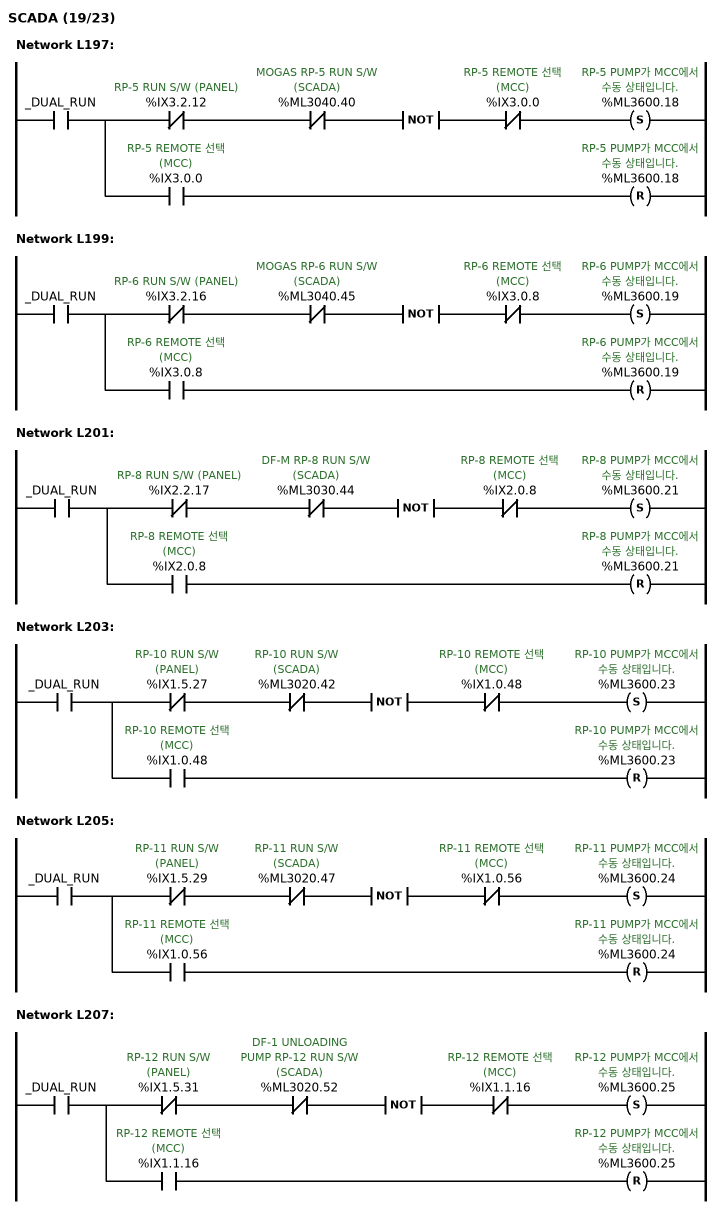
(* [picture p72: SCADA rungs L197-L207] *)
(* Rung L197 *)
IF NOT (_DUAL_RUN AND NOT %IX3.2.12 AND NOT %ML3040.40) AND NOT %IX3.0.0 THEN %ML3600.18 := TRUE; END_IF;
IF _DUAL_RUN AND %IX3.0.0 THEN %ML3600.18 := FALSE; END_IF;
(* Rung L199 *)
IF NOT (_DUAL_RUN AND NOT %IX3.2.16 AND NOT %ML3040.45) AND NOT %IX3.0.8 THEN %ML3600.19 := TRUE; END_IF;
IF _DUAL_RUN AND %IX3.0.8 THEN %ML3600.19 := FALSE; END_IF;
(* Rung L201 *)
IF NOT (_DUAL_RUN AND NOT %IX2.2.17 AND NOT %ML3030.44) AND NOT %IX2.0.8 THEN %ML3600.21 := TRUE; END_IF;
IF _DUAL_RUN AND %IX2.0.8 THEN %ML3600.21 := FALSE; END_IF;
(* Rung L203 *)
IF NOT (_DUAL_RUN AND NOT %IX1.5.27 AND NOT %ML3020.42) AND NOT %IX1.0.48 THEN %ML3600.23 := TRUE; END_IF;
IF _DUAL_RUN AND %IX1.0.48 THEN %ML3600.23 := FALSE; END_IF;
(* Rung L205 *)
IF NOT (_DUAL_RUN AND NOT %IX1.5.29 AND NOT %ML3020.47) AND NOT %IX1.0.56 THEN %ML3600.24 := TRUE; END_IF;
IF _DUAL_RUN AND %IX1.0.56 THEN %ML3600.24 := FALSE; END_IF;
(* Rung L207 *)
IF NOT (_DUAL_RUN AND NOT %IX1.5.31 AND NOT %ML3020.52) AND NOT %IX1.1.16 THEN %ML3600.25 := TRUE; END_IF;
IF _DUAL_RUN AND %IX1.1.16 THEN %ML3600.25 := FALSE; END_IF;

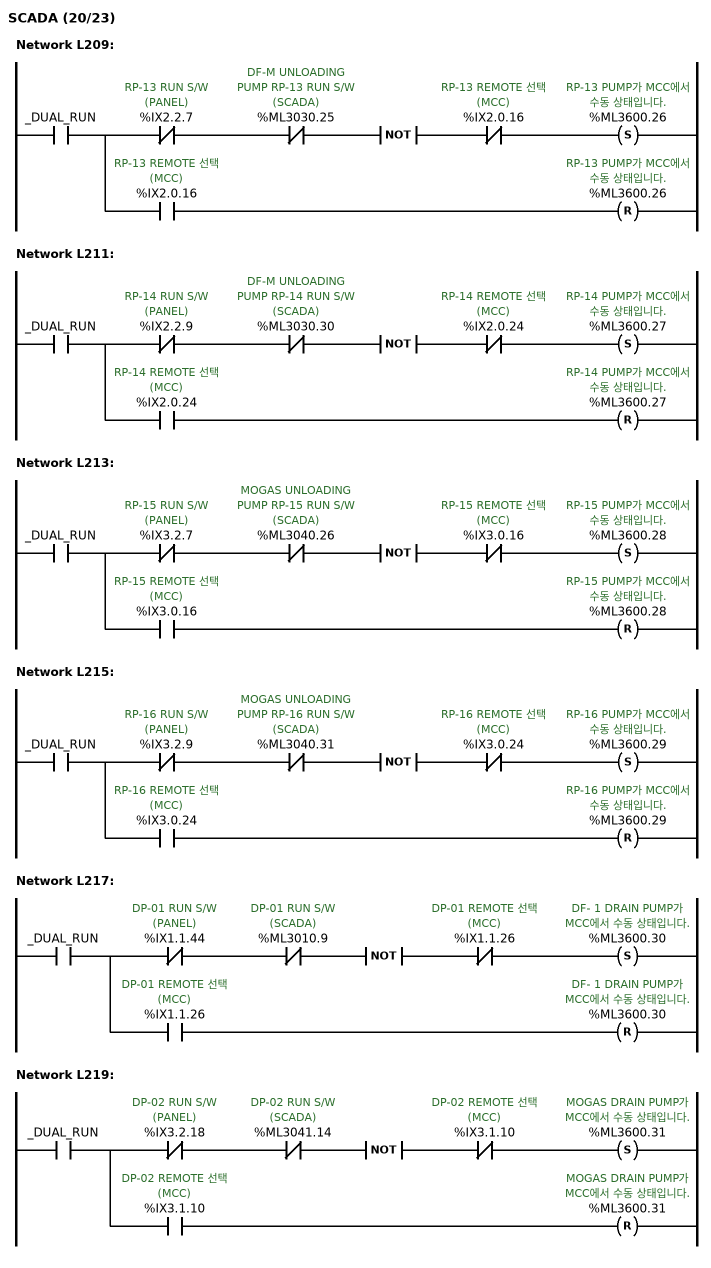
(* Rung L209 *)
IF NOT (_DUAL_RUN AND NOT %IX2.2.7 AND NOT %ML3030.25) AND NOT %IX2.0.16 THEN %ML3600.26 := TRUE; END_IF;
IF _DUAL_RUN AND %IX2.0.16 THEN %ML3600.26 := FALSE; END_IF;
(* Rung L211 *)
IF NOT (_DUAL_RUN AND NOT %IX2.2.9 AND NOT %ML3030.30) AND NOT %IX2.0.24 THEN %ML3600.27 := TRUE; END_IF;
IF _DUAL_RUN AND %IX2.0.24 THEN %ML3600.27 := FALSE; END_IF;
(* Rung L213 *)
IF NOT (_DUAL_RUN AND NOT %IX3.2.7 AND NOT %ML3040.26) AND NOT %IX3.0.16 THEN %ML3600.28 := TRUE; END_IF;
IF _DUAL_RUN AND %IX3.0.16 THEN %ML3600.28 := FALSE; END_IF;
(* Rung L215 *)
IF NOT (_DUAL_RUN AND NOT %IX3.2.9 AND NOT %ML3040.31) AND NOT %IX3.0.24 THEN %ML3600.29 := TRUE; END_IF;
IF _DUAL_RUN AND %IX3.0.24 THEN %ML3600.29 := FALSE; END_IF;
(* Rung L217 *)
IF NOT (_DUAL_RUN AND NOT %IX1.1.44 AND NOT %ML3010.9) AND NOT %IX1.1.26 THEN %ML3600.30 := TRUE; END_IF;
IF _DUAL_RUN AND %IX1.1.26 THEN %ML3600.30 := FALSE; END_IF;
(* Rung L219 *)
IF NOT (_DUAL_RUN AND NOT %IX3.2.18 AND NOT %ML3041.14) AND NOT %IX3.1.10 THEN %ML3600.31 := TRUE; END_IF;
IF _DUAL_RUN AND %IX3.1.10 THEN %ML3600.31 := FALSE; END_IF;

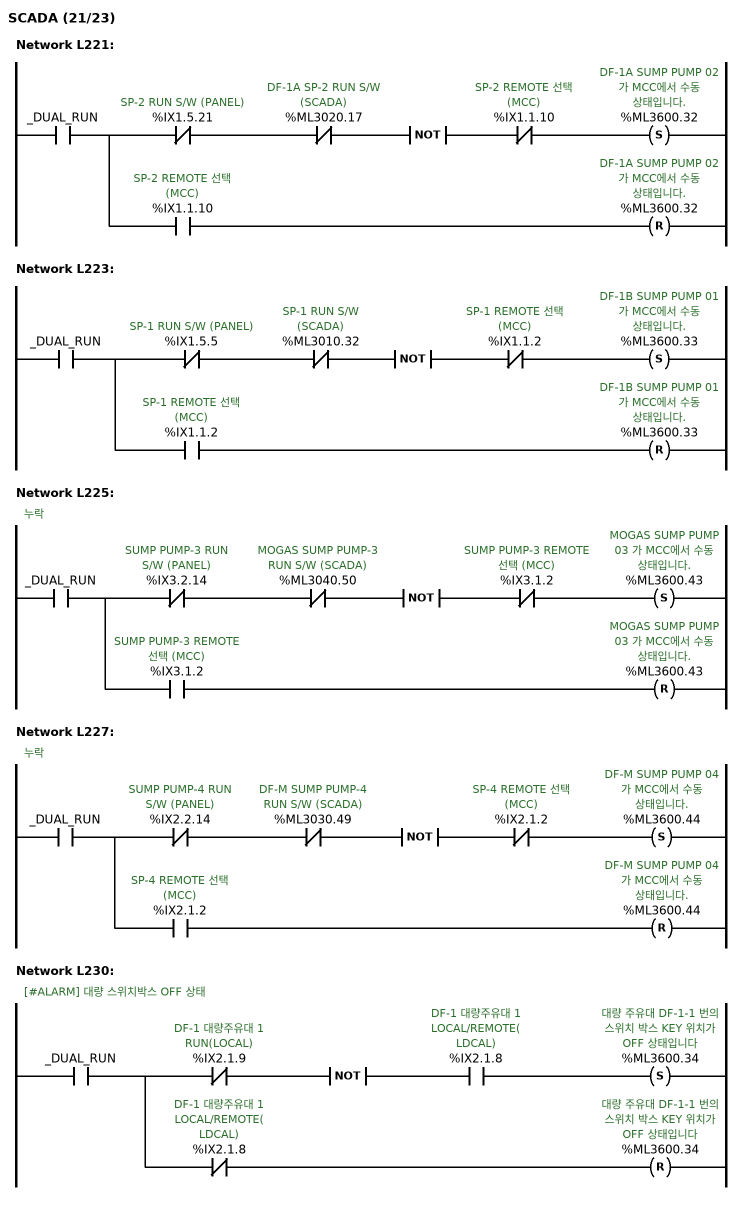
(* Rung L221 *)
IF NOT (_DUAL_RUN AND NOT %IX1.5.21 AND NOT %ML3020.17) AND NOT %IX1.1.10 THEN %ML3600.32 := TRUE; END_IF;
IF _DUAL_RUN AND %IX1.1.10 THEN %ML3600.32 := FALSE; END_IF;
(* Rung L223 *)
IF NOT (_DUAL_RUN AND NOT %IX1.5.5 AND NOT %ML3010.32) AND NOT %IX1.1.2 THEN %ML3600.33 := TRUE; END_IF;
IF _DUAL_RUN AND %IX1.1.2 THEN %ML3600.33 := FALSE; END_IF;
(* Rung L225 *)
IF NOT (_DUAL_RUN AND NOT %IX3.2.14 AND NOT %ML3040.50) AND NOT %IX3.1.2 THEN %ML3600.43 := TRUE; END_IF;
IF _DUAL_RUN AND %IX3.1.2 THEN %ML3600.43 := FALSE; END_IF;
(* 누락 *)
(* Rung L227 *)
IF NOT (_DUAL_RUN AND NOT %IX2.2.14 AND NOT %ML3030.49) AND NOT %IX2.1.2 THEN %ML3600.44 := TRUE; END_IF;
IF _DUAL_RUN AND %IX2.1.2 THEN %ML3600.44 := FALSE; END_IF;
(* 누락 *)
(* [#ALARM] 대량 스위치박스 OFF 상태 *)
(* Rung L230 *)
IF NOT (_DUAL_RUN AND NOT %IX2.1.9) AND %IX2.1.8 THEN %ML3600.34 := TRUE; END_IF;
IF _DUAL_RUN AND NOT %IX2.1.8 THEN %ML3600.34 := FALSE; END_IF;

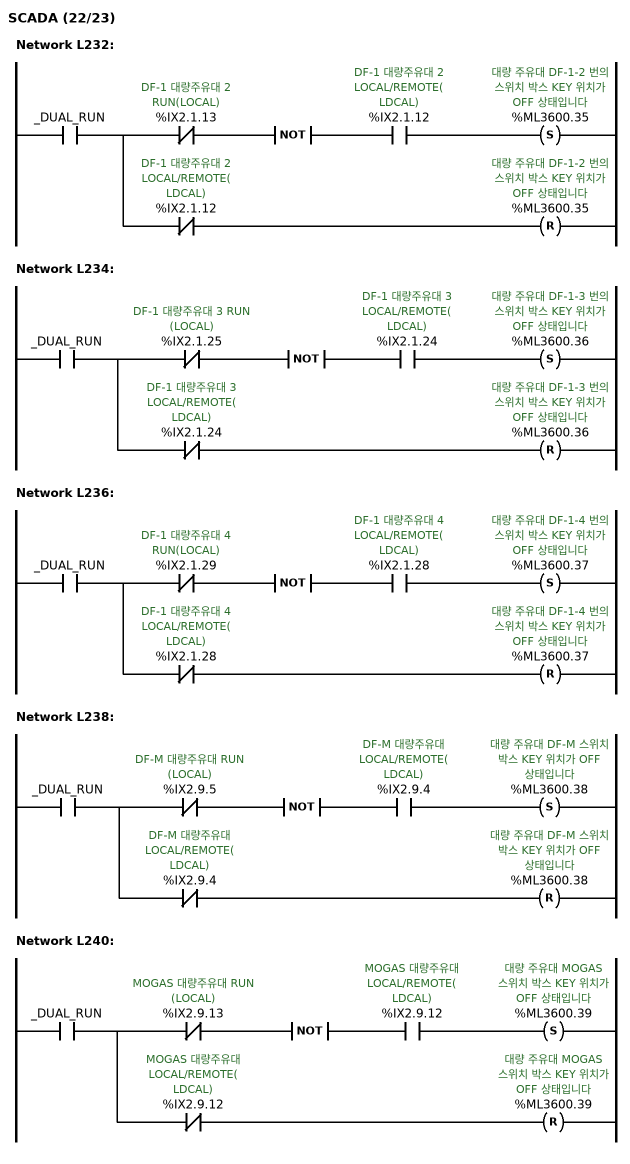
(* Rung L232 *)
IF NOT (_DUAL_RUN AND NOT %IX2.1.13) AND %IX2.1.12 THEN %ML3600.35 := TRUE; END_IF;
IF _DUAL_RUN AND NOT %IX2.1.12 THEN %ML3600.35 := FALSE; END_IF;
(* Rung L234 *)
IF NOT (_DUAL_RUN AND NOT %IX2.1.25) AND %IX2.1.24 THEN %ML3600.36 := TRUE; END_IF;
IF _DUAL_RUN AND NOT %IX2.1.24 THEN %ML3600.36 := FALSE; END_IF;
(* Rung L236 *)
IF NOT (_DUAL_RUN AND NOT %IX2.1.29) AND %IX2.1.28 THEN %ML3600.37 := TRUE; END_IF;
IF _DUAL_RUN AND NOT %IX2.1.28 THEN %ML3600.37 := FALSE; END_IF;
(* Rung L238 *)
IF NOT (_DUAL_RUN AND NOT %IX2.9.5) AND %IX2.9.4 THEN %ML3600.38 := TRUE; END_IF;
IF _DUAL_RUN AND NOT %IX2.9.4 THEN %ML3600.38 := FALSE; END_IF;
(* Rung L240 *)
IF NOT (_DUAL_RUN AND NOT %IX2.9.13) AND %IX2.9.12 THEN %ML3600.39 := TRUE; END_IF;
IF _DUAL_RUN AND NOT %IX2.9.12 THEN %ML3600.39 := FALSE; END_IF;

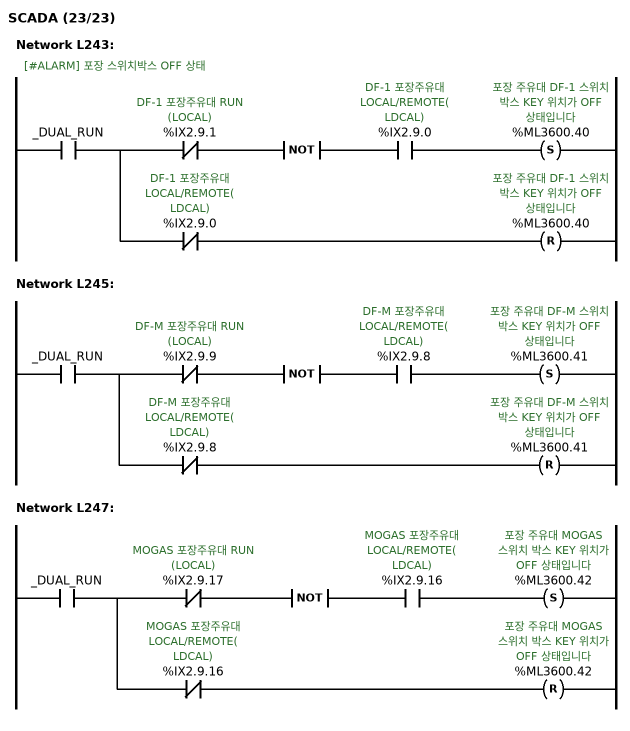
(* [#ALARM] 포장 스위치박스 OFF 상태 *)
(* Rung L243 *)
IF NOT (_DUAL_RUN AND NOT %IX2.9.1) AND %IX2.9.0 THEN %ML3600.40 := TRUE; END_IF;
IF _DUAL_RUN AND NOT %IX2.9.0 THEN %ML3600.40 := FALSE; END_IF;
(* Rung L245 *)
IF NOT (_DUAL_RUN AND NOT %IX2.9.9) AND %IX2.9.8 THEN %ML3600.41 := TRUE; END_IF;
IF _DUAL_RUN AND NOT %IX2.9.8 THEN %ML3600.41 := FALSE; END_IF;
(* Rung L247 *)
IF NOT (_DUAL_RUN AND NOT %IX2.9.17) AND %IX2.9.16 THEN %ML3600.42 := TRUE; END_IF;
IF _DUAL_RUN AND NOT %IX2.9.16 THEN %ML3600.42 := FALSE; END_IF;
END_PROGRAM

PROGRAM OUT (* task: 스캔 프로그램 *)
VAR
    D10 : BOOL;
    D1000 : BOOL;
    H16 : BOOL;
    INST : FF;
END_VAR
VAR
    _t1 : BOOL;
    _t2 : BOOL;
    _t3 : BOOL;
    _t4 : BOOL;
    _t5 : BOOL;
    _t6 : BOOL;
    _t7 : BOOL;
    _t8 : BOOL;
    _t9 : BOOL;
    _t10 : BOOL;
    _t11 : BOOL;
    _t12 : BOOL;
END_VAR

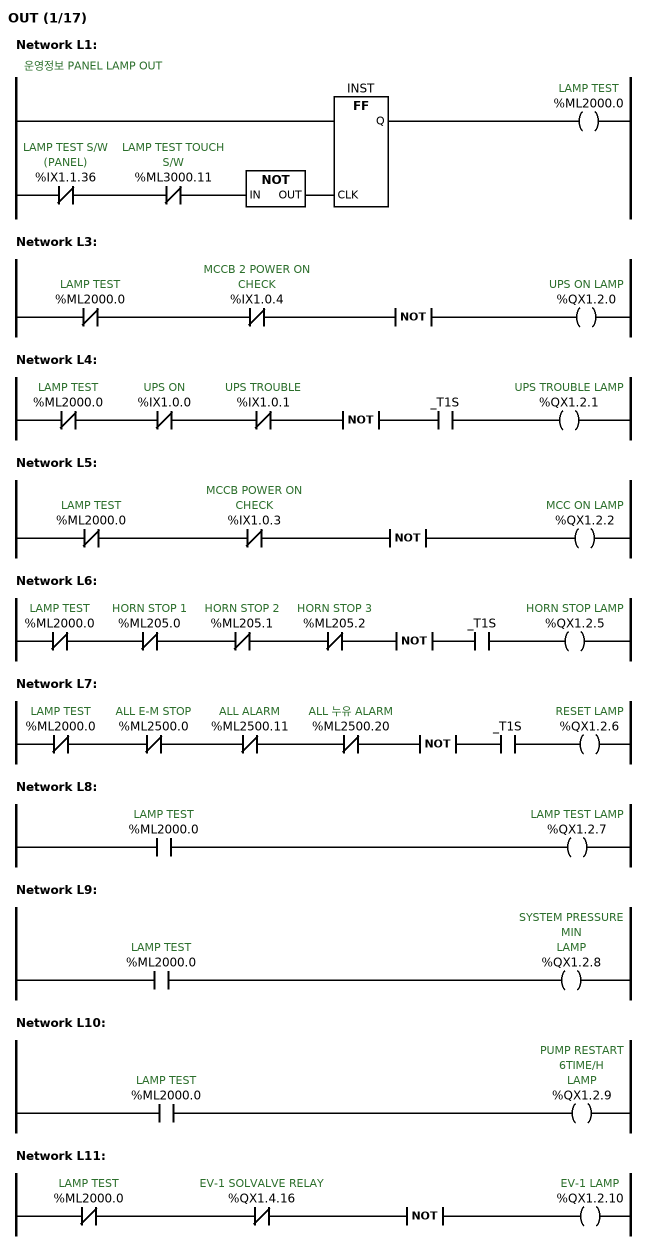
(* 운영정보 PANEL LAMP OUT *)
(* Rung L1 *)
INST(CLK := NOT (NOT %IX1.1.36 AND NOT %ML3000.11));
%ML2000.0 := INST.Q;
(* Rung L3 *)
%QX1.2.0 := NOT (NOT %ML2000.0 AND NOT %IX1.0.4);
(* Rung L4 *)
%QX1.2.1 := NOT (NOT %ML2000.0 AND NOT %IX1.0.0 AND NOT %IX1.0.1) AND _T1S;
(* Rung L5 *)
%QX1.2.2 := NOT (NOT %ML2000.0 AND NOT %IX1.0.3);
(* Rung L6 *)
%QX1.2.5 := NOT (NOT %ML2000.0 AND NOT %ML205.0 AND NOT %ML205.1 AND NOT %ML205.2) AND _T1S;
(* Rung L7 *)
%QX1.2.6 := NOT (NOT %ML2000.0 AND NOT %ML2500.0 AND NOT %ML2500.11 AND NOT %ML2500.20) AND _T1S;
(* Rung L8 *)
%QX1.2.7 := %ML2000.0;
(* Rung L9 *)
%QX1.2.8 := %ML2000.0;
(* Rung L10 *)
%QX1.2.9 := %ML2000.0;
(* Rung L11 *)
%QX1.2.10 := NOT (NOT %ML2000.0 AND NOT %QX1.4.16);

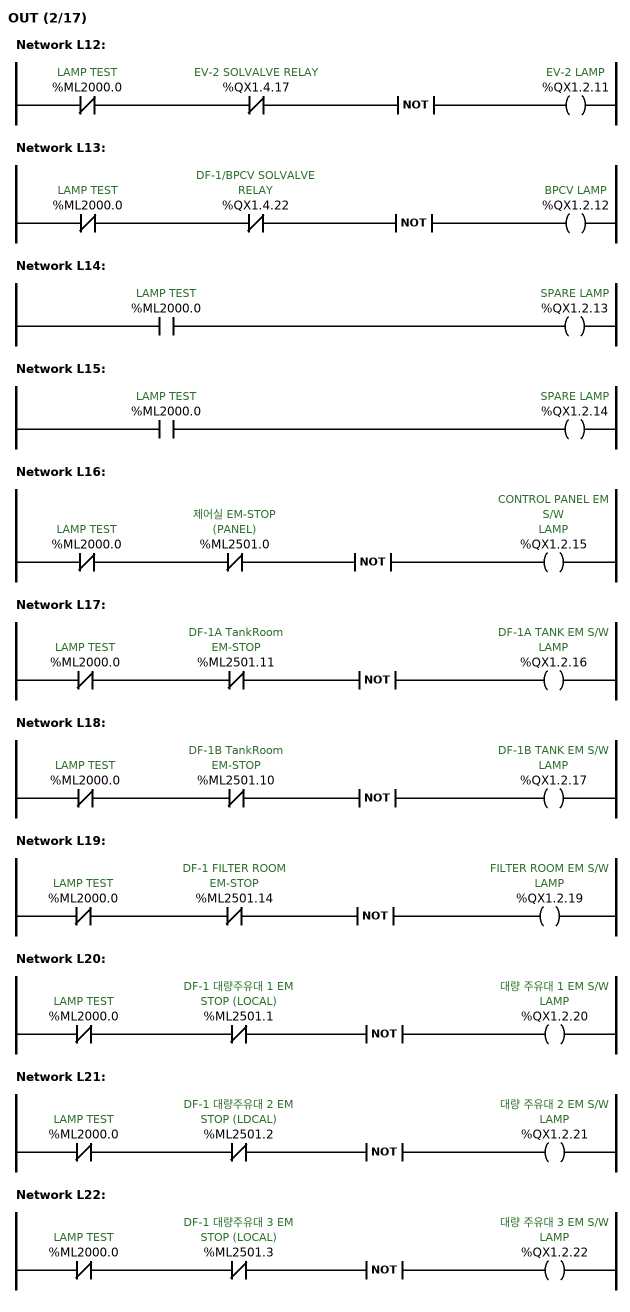
(* Rung L12 *)
%QX1.2.11 := NOT (NOT %ML2000.0 AND NOT %QX1.4.17);
(* Rung L13 *)
%QX1.2.12 := NOT (NOT %ML2000.0 AND NOT %QX1.4.22);
(* Rung L14 *)
%QX1.2.13 := %ML2000.0;
(* Rung L15 *)
%QX1.2.14 := %ML2000.0;
(* Rung L16 *)
%QX1.2.15 := NOT (NOT %ML2000.0 AND NOT %ML2501.0);
(* Rung L17 *)
%QX1.2.16 := NOT (NOT %ML2000.0 AND NOT %ML2501.11);
(* Rung L18 *)
%QX1.2.17 := NOT (NOT %ML2000.0 AND NOT %ML2501.10);
(* Rung L19 *)
%QX1.2.19 := NOT (NOT %ML2000.0 AND NOT %ML2501.14);
(* Rung L20 *)
%QX1.2.20 := NOT (NOT %ML2000.0 AND NOT %ML2501.1);
(* Rung L21 *)
%QX1.2.21 := NOT (NOT %ML2000.0 AND NOT %ML2501.2);
(* Rung L22 *)
%QX1.2.22 := NOT (NOT %ML2000.0 AND NOT %ML2501.3);

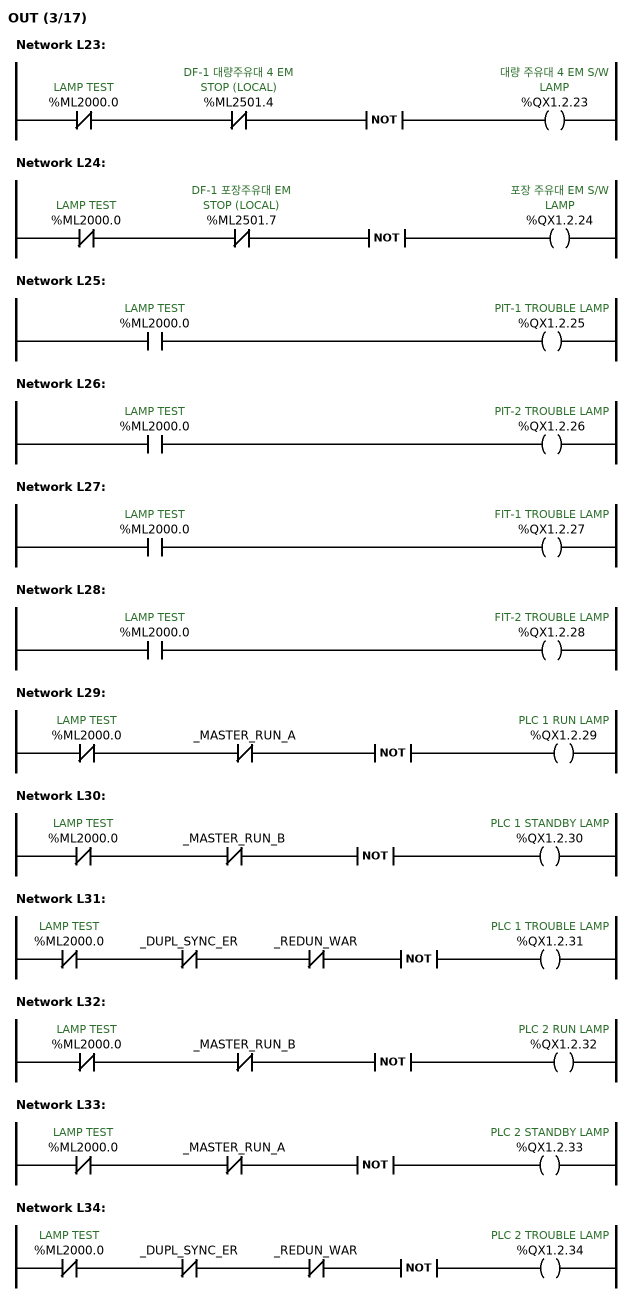
(* Rung L23 *)
%QX1.2.23 := NOT (NOT %ML2000.0 AND NOT %ML2501.4);
(* Rung L24 *)
%QX1.2.24 := NOT (NOT %ML2000.0 AND NOT %ML2501.7);
(* Rung L25 *)
%QX1.2.25 := %ML2000.0;
(* Rung L26 *)
%QX1.2.26 := %ML2000.0;
(* Rung L27 *)
%QX1.2.27 := %ML2000.0;
(* Rung L28 *)
%QX1.2.28 := %ML2000.0;
(* Rung L29 *)
%QX1.2.29 := NOT (NOT %ML2000.0 AND NOT _MASTER_RUN_A);
(* Rung L30 *)
%QX1.2.30 := NOT (NOT %ML2000.0 AND NOT _MASTER_RUN_B);
(* Rung L31 *)
%QX1.2.31 := NOT (NOT %ML2000.0 AND NOT _DUPL_SYNC_ER AND NOT _REDUN_WAR);
(* Rung L32 *)
%QX1.2.32 := NOT (NOT %ML2000.0 AND NOT _MASTER_RUN_B);
(* Rung L33 *)
%QX1.2.33 := NOT (NOT %ML2000.0 AND NOT _MASTER_RUN_A);
(* Rung L34 *)
%QX1.2.34 := NOT (NOT %ML2000.0 AND NOT _DUPL_SYNC_ER AND NOT _REDUN_WAR);

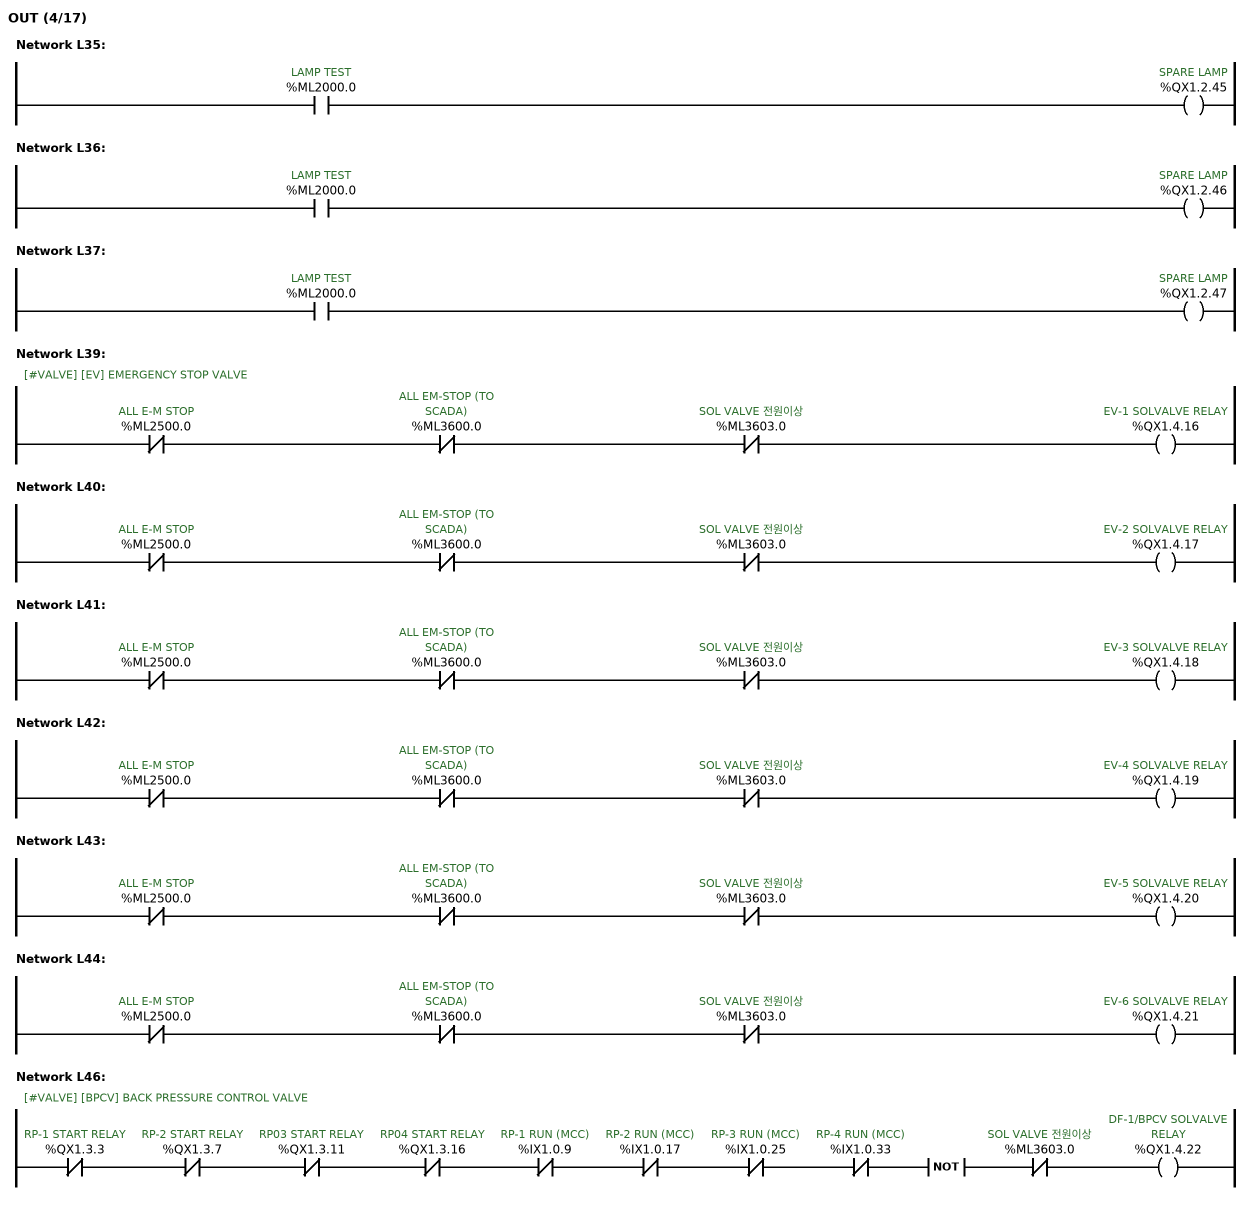
(* Rung L35 *)
%QX1.2.45 := %ML2000.0;
(* Rung L36 *)
%QX1.2.46 := %ML2000.0;
(* Rung L37 *)
%QX1.2.47 := %ML2000.0;
(* [#VALVE] [EV] EMERGENCY STOP VALVE *)
(* Rung L39 *)
%QX1.4.16 := NOT %ML2500.0 AND NOT %ML3600.0 AND NOT %ML3603.0;
(* Rung L40 *)
%QX1.4.17 := NOT %ML2500.0 AND NOT %ML3600.0 AND NOT %ML3603.0;
(* Rung L41 *)
%QX1.4.18 := NOT %ML2500.0 AND NOT %ML3600.0 AND NOT %ML3603.0;
(* Rung L42 *)
%QX1.4.19 := NOT %ML2500.0 AND NOT %ML3600.0 AND NOT %ML3603.0;
(* Rung L43 *)
%QX1.4.20 := NOT %ML2500.0 AND NOT %ML3600.0 AND NOT %ML3603.0;
(* Rung L44 *)
%QX1.4.21 := NOT %ML2500.0 AND NOT %ML3600.0 AND NOT %ML3603.0;
(* [#VALVE] [BPCV] BACK PRESSURE CONTROL VALVE *)
(* Rung L46 *)
%QX1.4.22 := NOT (NOT %QX1.3.3 AND NOT %QX1.3.7 AND NOT %QX1.3.11 AND NOT %QX1.3.16 AND NOT %IX1.0.9 AND NOT %IX1.0.17 AND NOT %IX1.0.25 AND NOT %IX1.0.33) AND NOT %ML3603.0;

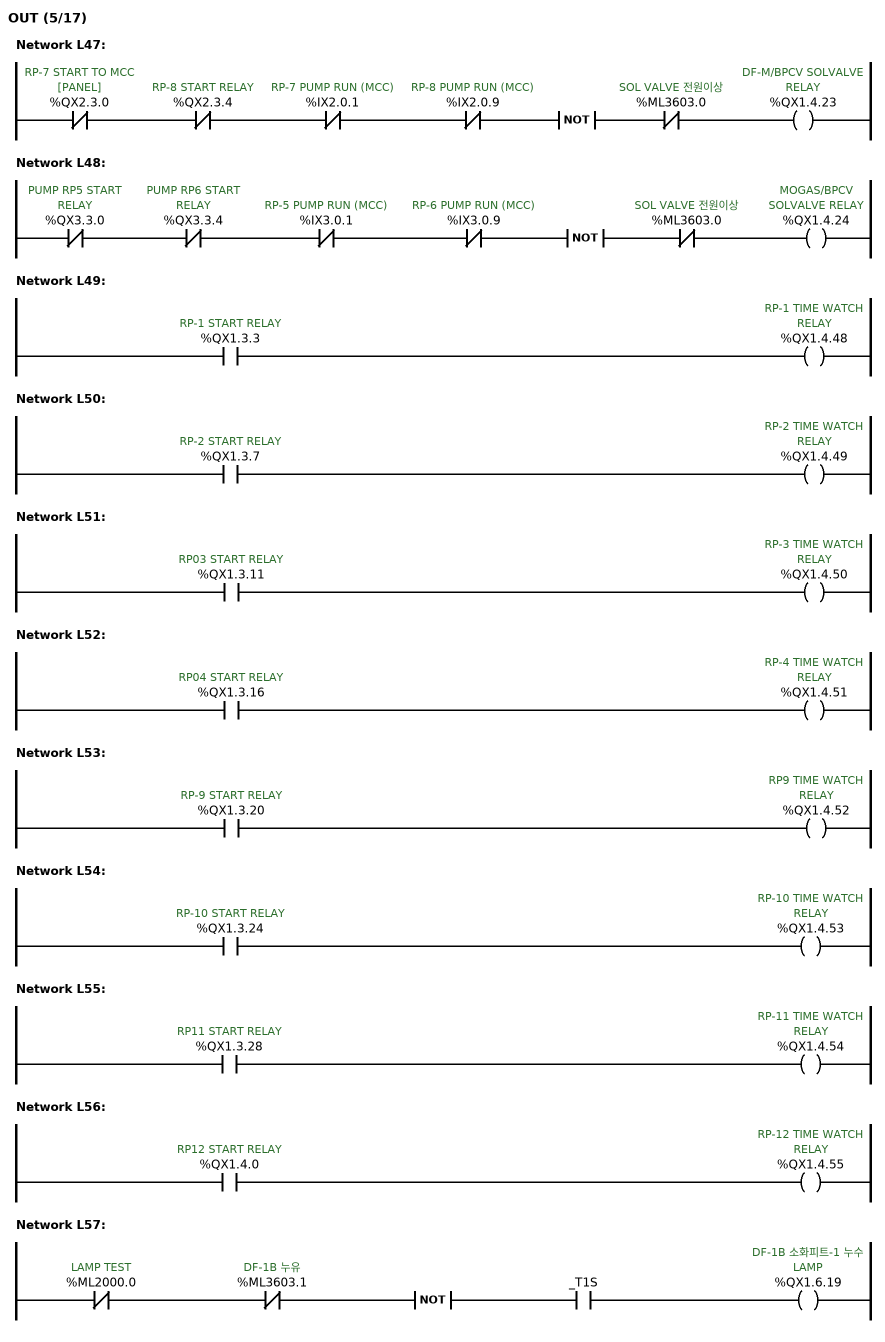
(* Rung L47 *)
%QX1.4.23 := NOT (NOT %QX2.3.0 AND NOT %QX2.3.4 AND NOT %IX2.0.1 AND NOT %IX2.0.9) AND NOT %ML3603.0;
(* Rung L48 *)
%QX1.4.24 := NOT (NOT %QX3.3.0 AND NOT %QX3.3.4 AND NOT %IX3.0.1 AND NOT %IX3.0.9) AND NOT %ML3603.0;
(* Rung L49 *)
%QX1.4.48 := %QX1.3.3;
(* Rung L50 *)
%QX1.4.49 := %QX1.3.7;
(* Rung L51 *)
%QX1.4.50 := %QX1.3.11;
(* Rung L52 *)
%QX1.4.51 := %QX1.3.16;
(* Rung L53 *)
%QX1.4.52 := %QX1.3.20;
(* Rung L54 *)
%QX1.4.53 := %QX1.3.24;
(* Rung L55 *)
%QX1.4.54 := %QX1.3.28;
(* Rung L56 *)
%QX1.4.55 := %QX1.4.0;
(* Rung L57 *)
%QX1.6.19 := NOT (NOT %ML2000.0 AND NOT %ML3603.1) AND _T1S;

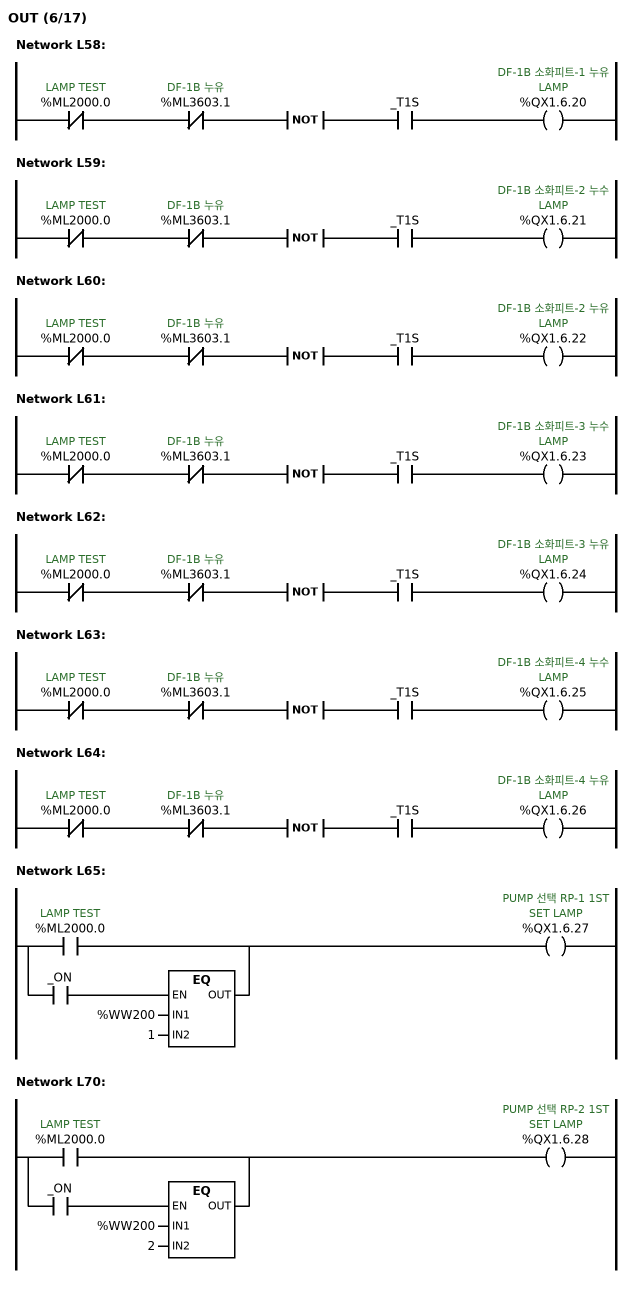
(* Rung L58 *)
%QX1.6.20 := NOT (NOT %ML2000.0 AND NOT %ML3603.1) AND _T1S;
(* Rung L59 *)
%QX1.6.21 := NOT (NOT %ML2000.0 AND NOT %ML3603.1) AND _T1S;
(* Rung L60 *)
%QX1.6.22 := NOT (NOT %ML2000.0 AND NOT %ML3603.1) AND _T1S;
(* Rung L61 *)
%QX1.6.23 := NOT (NOT %ML2000.0 AND NOT %ML3603.1) AND _T1S;
(* Rung L62 *)
%QX1.6.24 := NOT (NOT %ML2000.0 AND NOT %ML3603.1) AND _T1S;
(* Rung L63 *)
%QX1.6.25 := NOT (NOT %ML2000.0 AND NOT %ML3603.1) AND _T1S;
(* Rung L64 *)
%QX1.6.26 := NOT (NOT %ML2000.0 AND NOT %ML3603.1) AND _T1S;
(* Rung L65 *)
IF _ON THEN _t1 := %WW200 = 1; END_IF;
%QX1.6.27 := %ML2000.0 OR _t1;
(* Rung L70 *)
IF _ON THEN _t2 := %WW200 = 2; END_IF;
%QX1.6.28 := %ML2000.0 OR _t2;

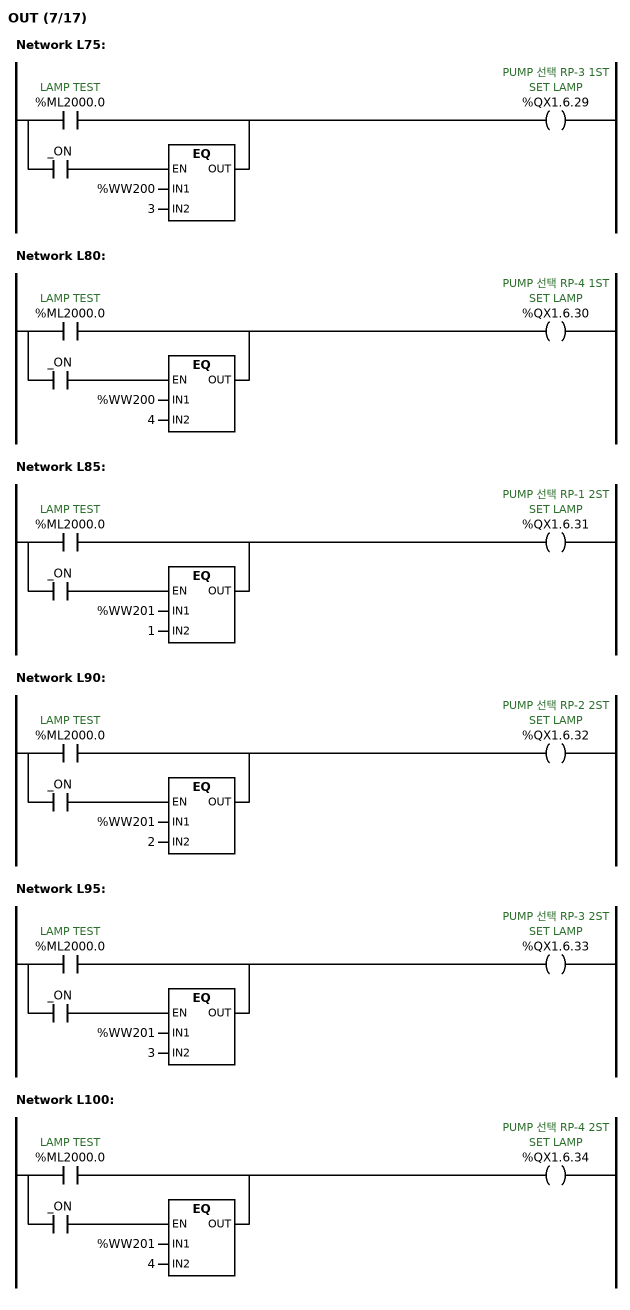
(* Rung L75 *)
IF _ON THEN _t3 := %WW200 = 3; END_IF;
%QX1.6.29 := %ML2000.0 OR _t3;
(* Rung L80 *)
IF _ON THEN _t4 := %WW200 = 4; END_IF;
%QX1.6.30 := %ML2000.0 OR _t4;
(* Rung L85 *)
IF _ON THEN _t5 := %WW201 = 1; END_IF;
%QX1.6.31 := %ML2000.0 OR _t5;
(* Rung L90 *)
IF _ON THEN _t6 := %WW201 = 2; END_IF;
%QX1.6.32 := %ML2000.0 OR _t6;
(* Rung L95 *)
IF _ON THEN _t7 := %WW201 = 3; END_IF;
%QX1.6.33 := %ML2000.0 OR _t7;
(* Rung L100 *)
IF _ON THEN _t8 := %WW201 = 4; END_IF;
%QX1.6.34 := %ML2000.0 OR _t8;

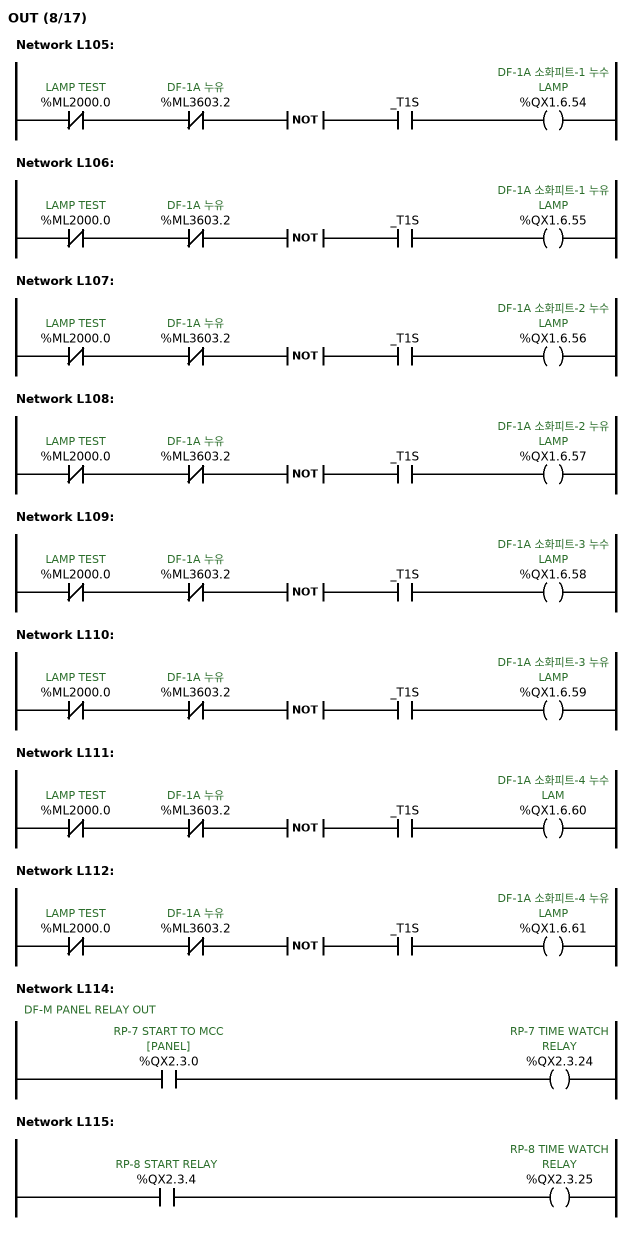
(* Rung L105 *)
%QX1.6.54 := NOT (NOT %ML2000.0 AND NOT %ML3603.2) AND _T1S;
(* Rung L106 *)
%QX1.6.55 := NOT (NOT %ML2000.0 AND NOT %ML3603.2) AND _T1S;
(* Rung L107 *)
%QX1.6.56 := NOT (NOT %ML2000.0 AND NOT %ML3603.2) AND _T1S;
(* Rung L108 *)
%QX1.6.57 := NOT (NOT %ML2000.0 AND NOT %ML3603.2) AND _T1S;
(* Rung L109 *)
%QX1.6.58 := NOT (NOT %ML2000.0 AND NOT %ML3603.2) AND _T1S;
(* Rung L110 *)
%QX1.6.59 := NOT (NOT %ML2000.0 AND NOT %ML3603.2) AND _T1S;
(* Rung L111 *)
%QX1.6.60 := NOT (NOT %ML2000.0 AND NOT %ML3603.2) AND _T1S;
(* Rung L112 *)
%QX1.6.61 := NOT (NOT %ML2000.0 AND NOT %ML3603.2) AND _T1S;
(* DF-M PANEL RELAY OUT *)
(* Rung L114 *)
%QX2.3.24 := %QX2.3.0;
(* Rung L115 *)
%QX2.3.25 := %QX2.3.4;

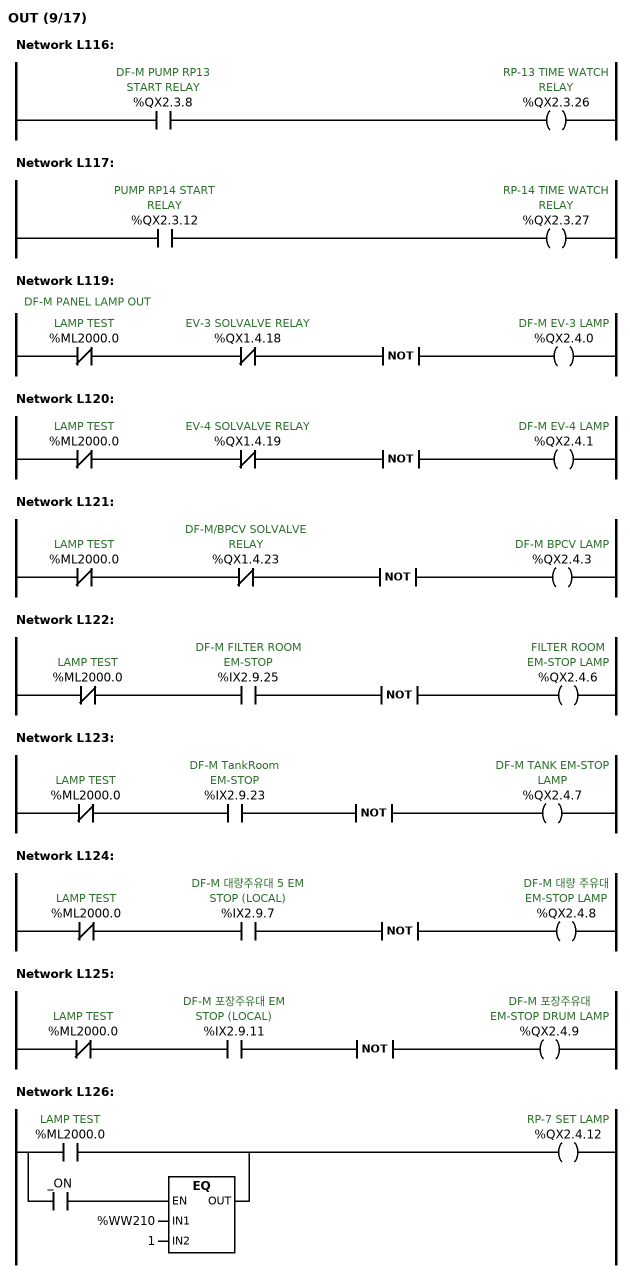
(* Rung L116 *)
%QX2.3.26 := %QX2.3.8;
(* Rung L117 *)
%QX2.3.27 := %QX2.3.12;
(* DF-M PANEL LAMP OUT *)
(* Rung L119 *)
%QX2.4.0 := NOT (NOT %ML2000.0 AND NOT %QX1.4.18);
(* Rung L120 *)
%QX2.4.1 := NOT (NOT %ML2000.0 AND NOT %QX1.4.19);
(* Rung L121 *)
%QX2.4.3 := NOT (NOT %ML2000.0 AND NOT %QX1.4.23);
(* Rung L122 *)
%QX2.4.6 := NOT (NOT %ML2000.0 AND %IX2.9.25);
(* Rung L123 *)
%QX2.4.7 := NOT (NOT %ML2000.0 AND %IX2.9.23);
(* Rung L124 *)
%QX2.4.8 := NOT (NOT %ML2000.0 AND %IX2.9.7);
(* Rung L125 *)
%QX2.4.9 := NOT (NOT %ML2000.0 AND %IX2.9.11);
(* Rung L126 *)
IF _ON THEN _t9 := %WW210 = 1; END_IF;
%QX2.4.12 := %ML2000.0 OR _t9;

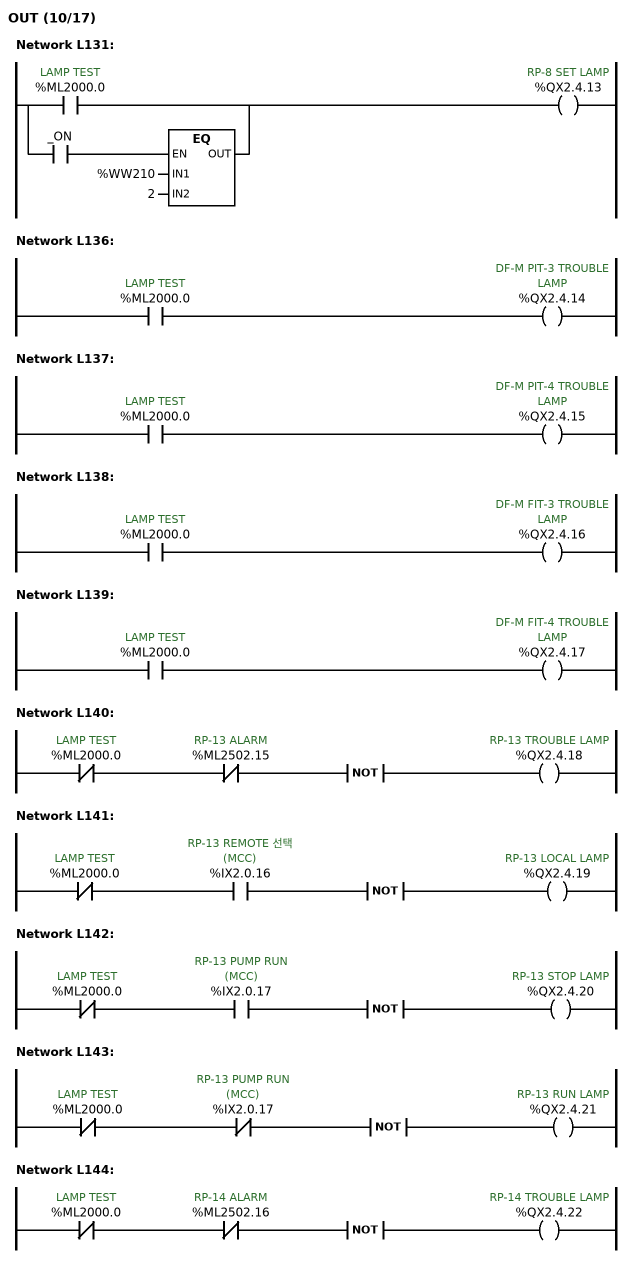
(* Rung L131 *)
IF _ON THEN _t10 := %WW210 = 2; END_IF;
%QX2.4.13 := %ML2000.0 OR _t10;
(* Rung L136 *)
%QX2.4.14 := %ML2000.0;
(* Rung L137 *)
%QX2.4.15 := %ML2000.0;
(* Rung L138 *)
%QX2.4.16 := %ML2000.0;
(* Rung L139 *)
%QX2.4.17 := %ML2000.0;
(* Rung L140 *)
%QX2.4.18 := NOT (NOT %ML2000.0 AND NOT %ML2502.15);
(* Rung L141 *)
%QX2.4.19 := NOT (NOT %ML2000.0 AND %IX2.0.16);
(* Rung L142 *)
%QX2.4.20 := NOT (NOT %ML2000.0 AND %IX2.0.17);
(* Rung L143 *)
%QX2.4.21 := NOT (NOT %ML2000.0 AND NOT %IX2.0.17);
(* Rung L144 *)
%QX2.4.22 := NOT (NOT %ML2000.0 AND NOT %ML2502.16);

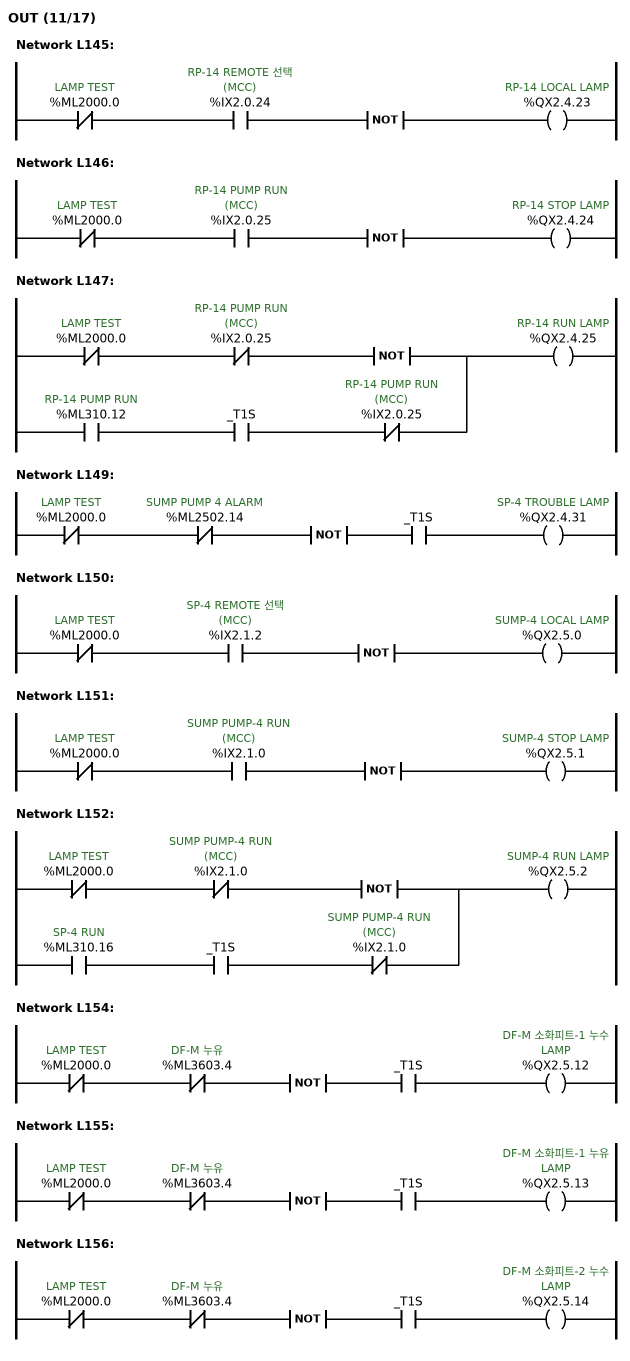
(* Rung L145 *)
%QX2.4.23 := NOT (NOT %ML2000.0 AND %IX2.0.24);
(* Rung L146 *)
%QX2.4.24 := NOT (NOT %ML2000.0 AND %IX2.0.25);
(* Rung L147 *)
%QX2.4.25 := NOT (NOT %ML2000.0 AND NOT %IX2.0.25) OR (%ML310.12 AND _T1S AND NOT %IX2.0.25);
(* Rung L149 *)
%QX2.4.31 := NOT (NOT %ML2000.0 AND NOT %ML2502.14) AND _T1S;
(* Rung L150 *)
%QX2.5.0 := NOT (NOT %ML2000.0 AND %IX2.1.2);
(* Rung L151 *)
%QX2.5.1 := NOT (NOT %ML2000.0 AND %IX2.1.0);
(* Rung L152 *)
%QX2.5.2 := NOT (NOT %ML2000.0 AND NOT %IX2.1.0) OR (%ML310.16 AND _T1S AND NOT %IX2.1.0);
(* Rung L154 *)
%QX2.5.12 := NOT (NOT %ML2000.0 AND NOT %ML3603.4) AND _T1S;
(* Rung L155 *)
%QX2.5.13 := NOT (NOT %ML2000.0 AND NOT %ML3603.4) AND _T1S;
(* Rung L156 *)
%QX2.5.14 := NOT (NOT %ML2000.0 AND NOT %ML3603.4) AND _T1S;

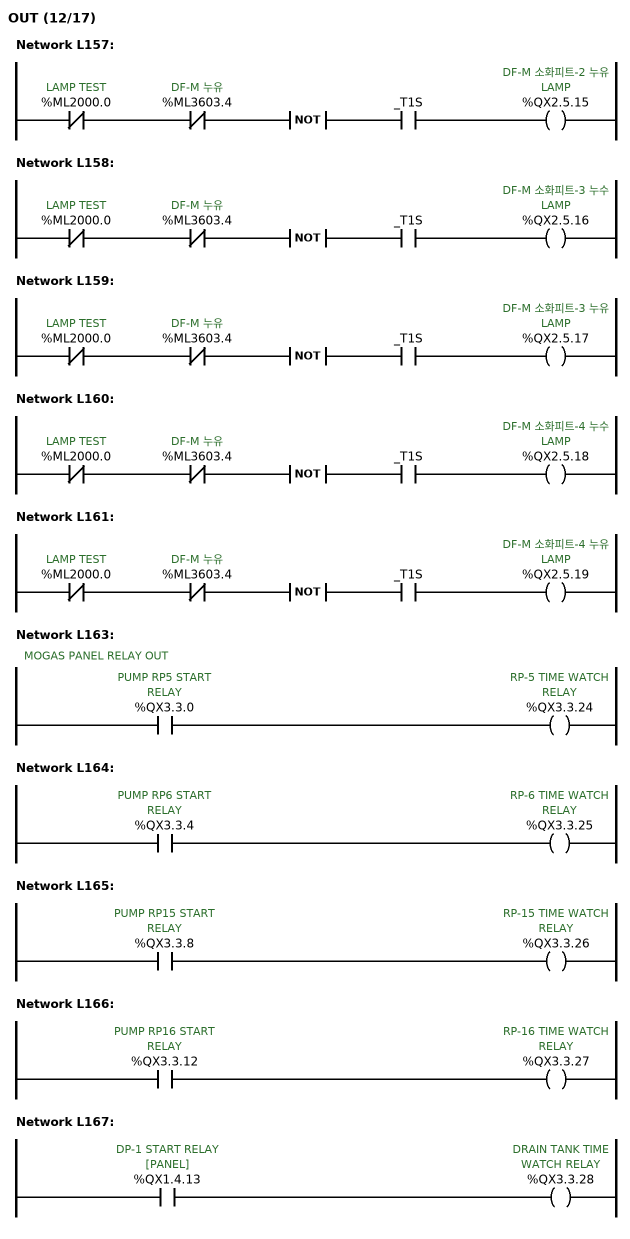
(* Rung L157 *)
%QX2.5.15 := NOT (NOT %ML2000.0 AND NOT %ML3603.4) AND _T1S;
(* Rung L158 *)
%QX2.5.16 := NOT (NOT %ML2000.0 AND NOT %ML3603.4) AND _T1S;
(* Rung L159 *)
%QX2.5.17 := NOT (NOT %ML2000.0 AND NOT %ML3603.4) AND _T1S;
(* Rung L160 *)
%QX2.5.18 := NOT (NOT %ML2000.0 AND NOT %ML3603.4) AND _T1S;
(* Rung L161 *)
%QX2.5.19 := NOT (NOT %ML2000.0 AND NOT %ML3603.4) AND _T1S;
(* MOGAS PANEL RELAY OUT *)
(* Rung L163 *)
%QX3.3.24 := %QX3.3.0;
(* Rung L164 *)
%QX3.3.25 := %QX3.3.4;
(* Rung L165 *)
%QX3.3.26 := %QX3.3.8;
(* Rung L166 *)
%QX3.3.27 := %QX3.3.12;
(* Rung L167 *)
%QX3.3.28 := %QX1.4.13;

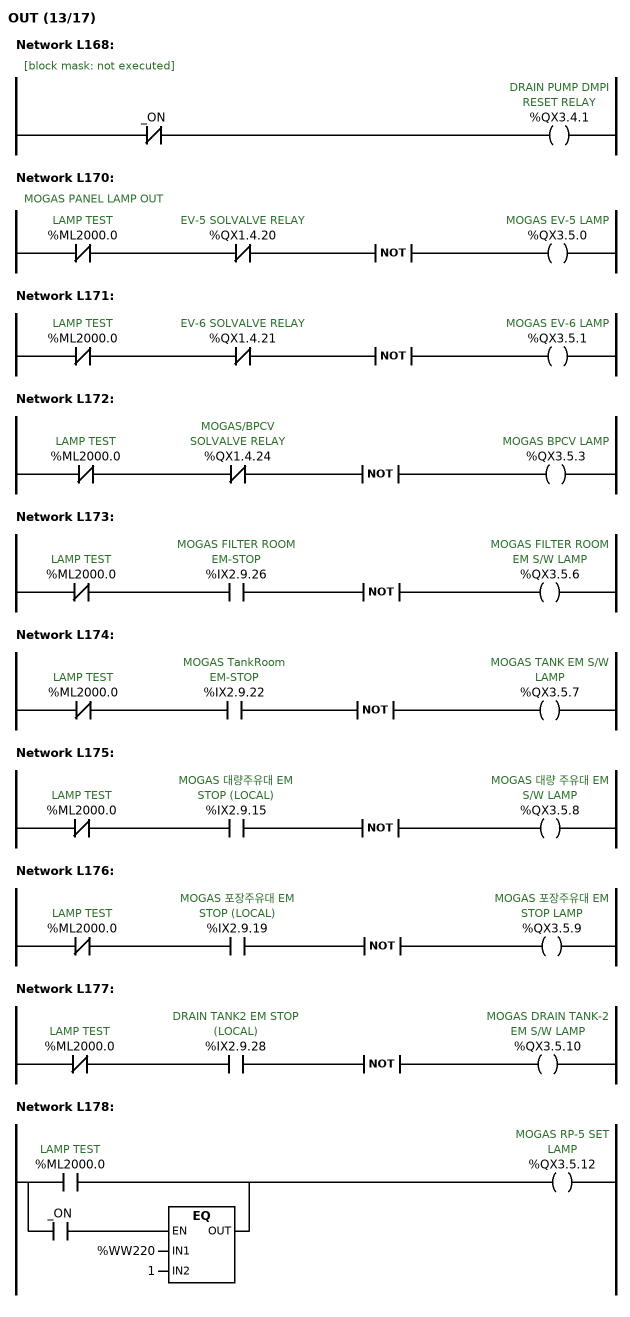
(* Rung L168 is block-masked: not executed *)
// %QX3.4.1 := NOT _ON;
(* MOGAS PANEL LAMP OUT *)
(* Rung L170 *)
%QX3.5.0 := NOT (NOT %ML2000.0 AND NOT %QX1.4.20);
(* Rung L171 *)
%QX3.5.1 := NOT (NOT %ML2000.0 AND NOT %QX1.4.21);
(* Rung L172 *)
%QX3.5.3 := NOT (NOT %ML2000.0 AND NOT %QX1.4.24);
(* Rung L173 *)
%QX3.5.6 := NOT (NOT %ML2000.0 AND %IX2.9.26);
(* Rung L174 *)
%QX3.5.7 := NOT (NOT %ML2000.0 AND %IX2.9.22);
(* Rung L175 *)
%QX3.5.8 := NOT (NOT %ML2000.0 AND %IX2.9.15);
(* Rung L176 *)
%QX3.5.9 := NOT (NOT %ML2000.0 AND %IX2.9.19);
(* Rung L177 *)
%QX3.5.10 := NOT (NOT %ML2000.0 AND %IX2.9.28);
(* Rung L178 *)
IF _ON THEN _t11 := %WW220 = 1; END_IF;
%QX3.5.12 := %ML2000.0 OR _t11;

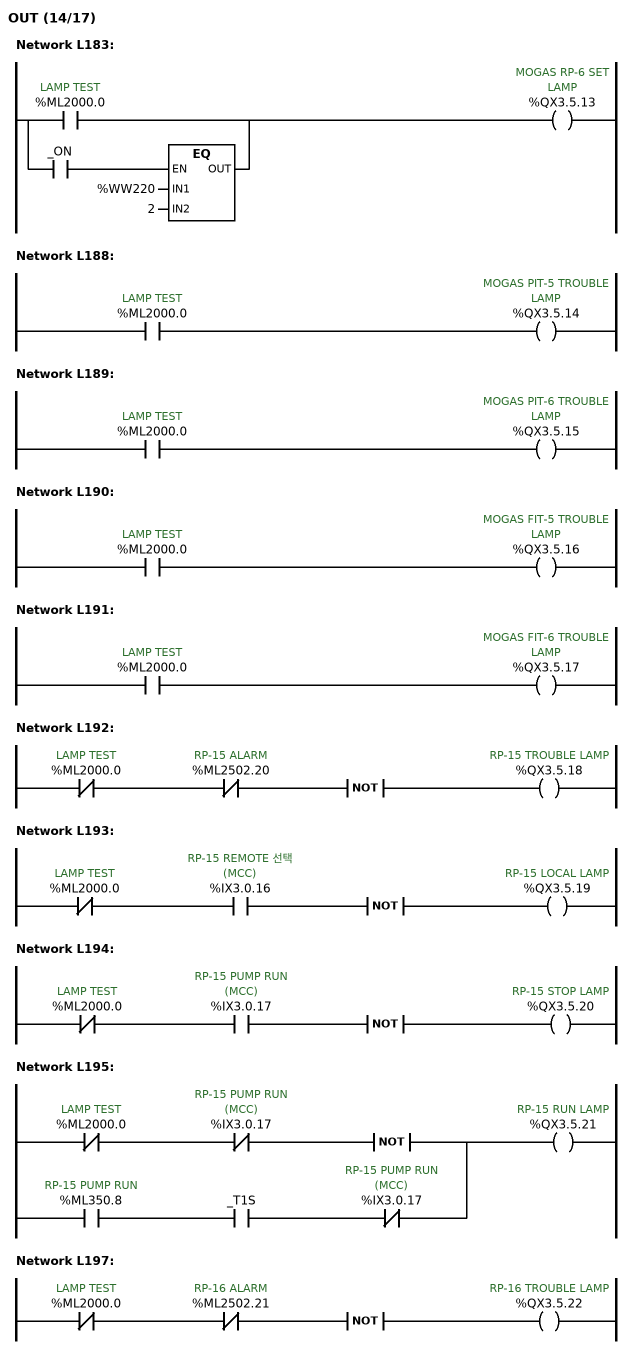
(* Rung L183 *)
IF _ON THEN _t12 := %WW220 = 2; END_IF;
%QX3.5.13 := %ML2000.0 OR _t12;
(* Rung L188 *)
%QX3.5.14 := %ML2000.0;
(* Rung L189 *)
%QX3.5.15 := %ML2000.0;
(* Rung L190 *)
%QX3.5.16 := %ML2000.0;
(* Rung L191 *)
%QX3.5.17 := %ML2000.0;
(* Rung L192 *)
%QX3.5.18 := NOT (NOT %ML2000.0 AND NOT %ML2502.20);
(* Rung L193 *)
%QX3.5.19 := NOT (NOT %ML2000.0 AND %IX3.0.16);
(* Rung L194 *)
%QX3.5.20 := NOT (NOT %ML2000.0 AND %IX3.0.17);
(* Rung L195 *)
%QX3.5.21 := NOT (NOT %ML2000.0 AND NOT %IX3.0.17) OR (%ML350.8 AND _T1S AND NOT %IX3.0.17);
(* Rung L197 *)
%QX3.5.22 := NOT (NOT %ML2000.0 AND NOT %ML2502.21);

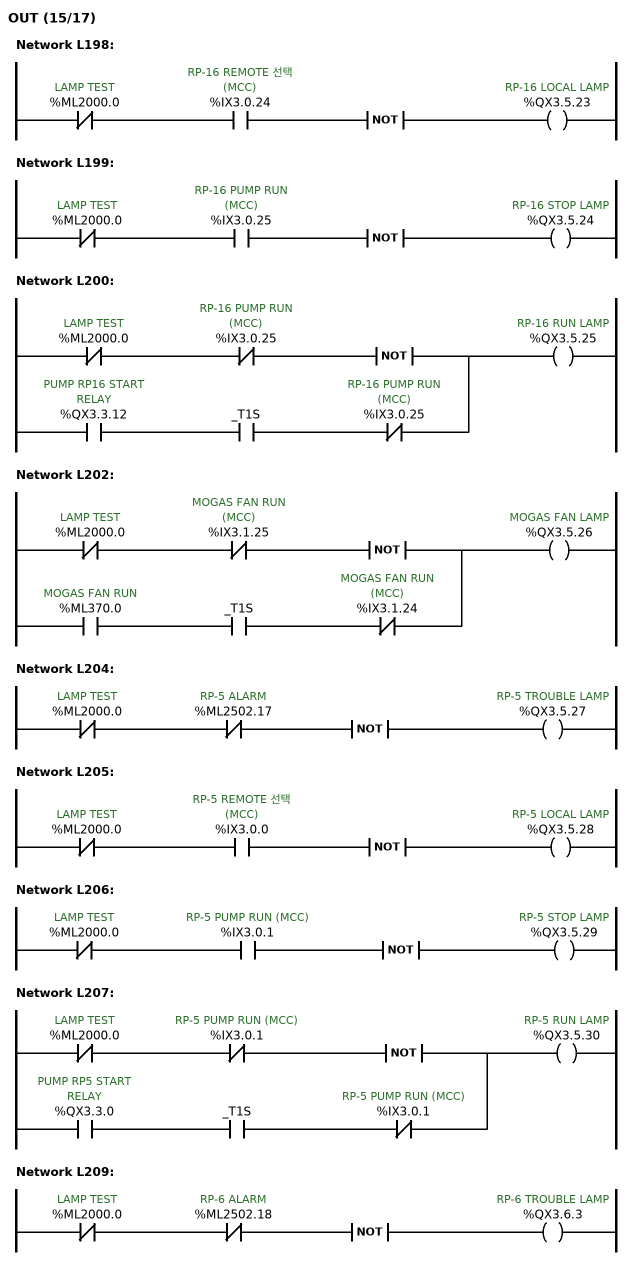
(* Rung L198 *)
%QX3.5.23 := NOT (NOT %ML2000.0 AND %IX3.0.24);
(* Rung L199 *)
%QX3.5.24 := NOT (NOT %ML2000.0 AND %IX3.0.25);
(* Rung L200 *)
%QX3.5.25 := NOT (NOT %ML2000.0 AND NOT %IX3.0.25) OR (%QX3.3.12 AND _T1S AND NOT %IX3.0.25);
(* Rung L202 *)
%QX3.5.26 := NOT (NOT %ML2000.0 AND NOT %IX3.1.25) OR (%ML370.0 AND _T1S AND NOT %IX3.1.24);
(* Rung L204 *)
%QX3.5.27 := NOT (NOT %ML2000.0 AND NOT %ML2502.17);
(* Rung L205 *)
%QX3.5.28 := NOT (NOT %ML2000.0 AND %IX3.0.0);
(* Rung L206 *)
%QX3.5.29 := NOT (NOT %ML2000.0 AND %IX3.0.1);
(* Rung L207 *)
%QX3.5.30 := NOT (NOT %ML2000.0 AND NOT %IX3.0.1) OR (%QX3.3.0 AND _T1S AND NOT %IX3.0.1);
(* Rung L209 *)
%QX3.6.3 := NOT (NOT %ML2000.0 AND NOT %ML2502.18);

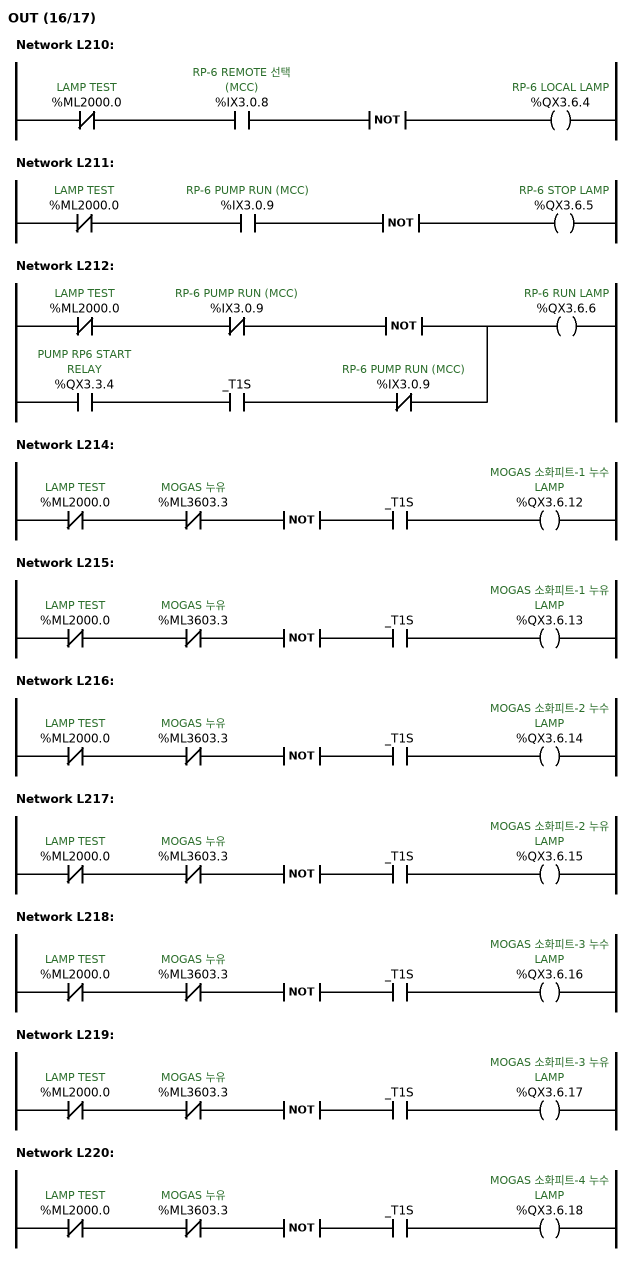
(* Rung L210 *)
%QX3.6.4 := NOT (NOT %ML2000.0 AND %IX3.0.8);
(* Rung L211 *)
%QX3.6.5 := NOT (NOT %ML2000.0 AND %IX3.0.9);
(* Rung L212 *)
%QX3.6.6 := NOT (NOT %ML2000.0 AND NOT %IX3.0.9) OR (%QX3.3.4 AND _T1S AND NOT %IX3.0.9);
(* Rung L214 *)
%QX3.6.12 := NOT (NOT %ML2000.0 AND NOT %ML3603.3) AND _T1S;
(* Rung L215 *)
%QX3.6.13 := NOT (NOT %ML2000.0 AND NOT %ML3603.3) AND _T1S;
(* Rung L216 *)
%QX3.6.14 := NOT (NOT %ML2000.0 AND NOT %ML3603.3) AND _T1S;
(* Rung L217 *)
%QX3.6.15 := NOT (NOT %ML2000.0 AND NOT %ML3603.3) AND _T1S;
(* Rung L218 *)
%QX3.6.16 := NOT (NOT %ML2000.0 AND NOT %ML3603.3) AND _T1S;
(* Rung L219 *)
%QX3.6.17 := NOT (NOT %ML2000.0 AND NOT %ML3603.3) AND _T1S;
(* Rung L220 *)
%QX3.6.18 := NOT (NOT %ML2000.0 AND NOT %ML3603.3) AND _T1S;

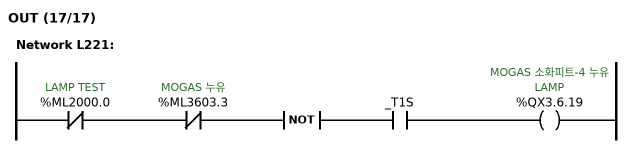
(* Rung L221 *)
%QX3.6.19 := NOT (NOT %ML2000.0 AND NOT %ML3603.3) AND _T1S;
END_PROGRAM

PROGRAM ALARM (* task: 스캔 프로그램 *)

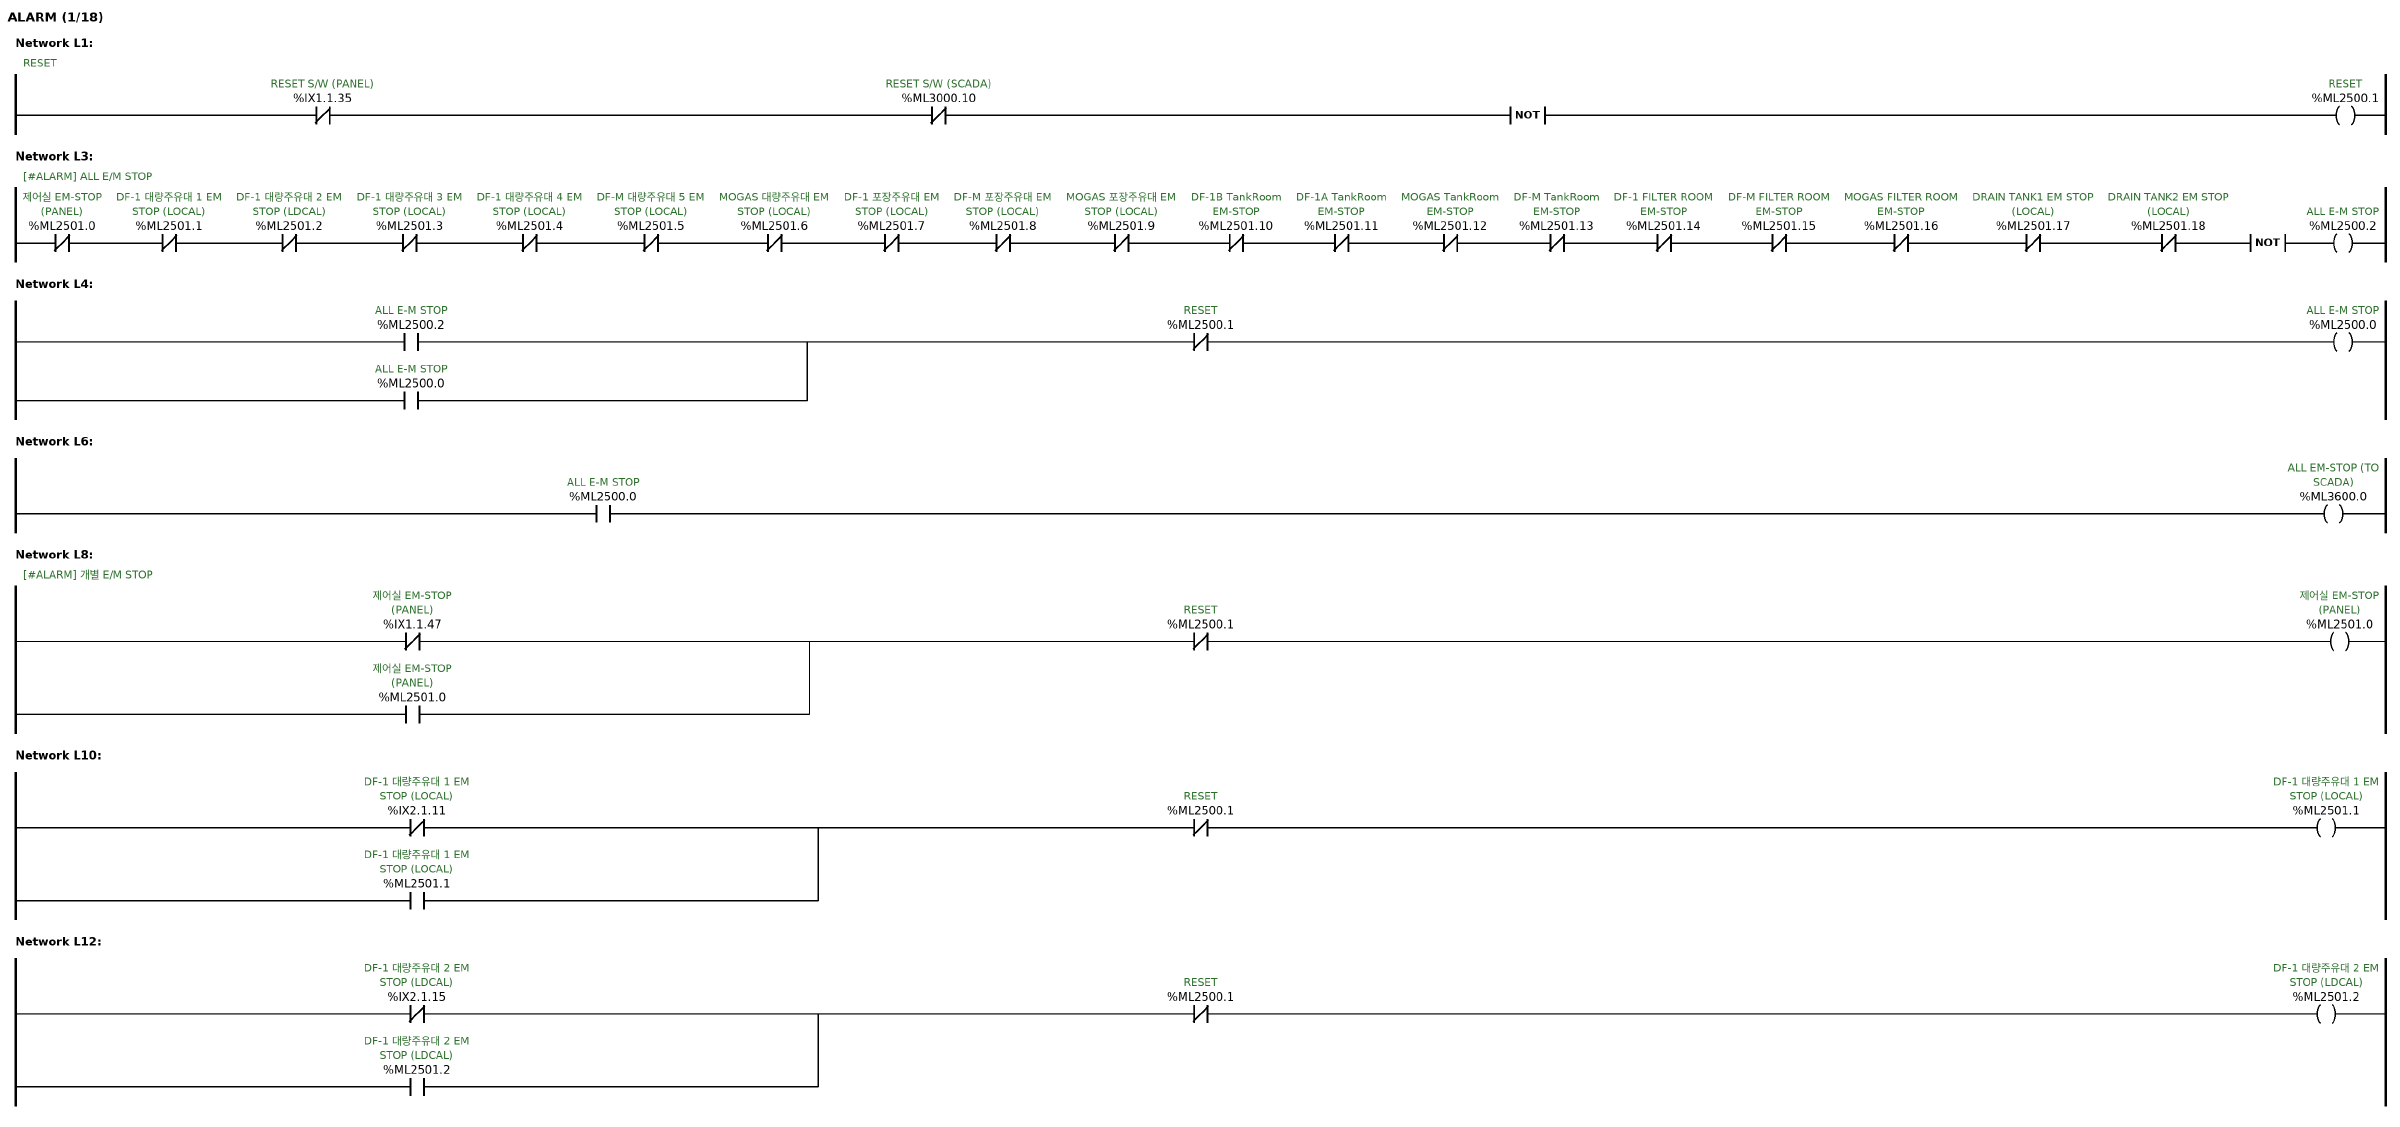
(* RESET *)
(* Rung L1 *)
%ML2500.1 := NOT (NOT %IX1.1.35 AND NOT %ML3000.10);
(* [#ALARM] ALL E/M STOP *)
(* Rung L3 *)
%ML2500.2 := NOT (NOT %ML2501.0 AND NOT %ML2501.1 AND NOT %ML2501.2 AND NOT %ML2501.3 AND NOT %ML2501.4 AND NOT %ML2501.5 AND NOT %ML2501.6 AND NOT %ML2501.7 AND NOT %ML2501.8 AND NOT %ML2501.9 AND NOT %ML2501.10 AND NOT %ML2501.11 AND NOT %ML2501.12 AND NOT %ML2501.13 AND NOT %ML2501.14 AND NOT %ML2501.15 AND NOT %ML2501.16 AND NOT %ML2501.17 AND NOT %ML2501.18);
(* Rung L4 *)
%ML2500.0 := (%ML2500.2 OR %ML2500.0) AND NOT %ML2500.1;
(* Rung L6 *)
%ML3600.0 := %ML2500.0;
(* [#ALARM] 개별 E/M STOP *)
(* Rung L8 *)
%ML2501.0 := (NOT %IX1.1.47 OR %ML2501.0) AND NOT %ML2500.1;
(* Rung L10 *)
%ML2501.1 := (NOT %IX2.1.11 OR %ML2501.1) AND NOT %ML2500.1;
(* Rung L12 *)
%ML2501.2 := (NOT %IX2.1.15 OR %ML2501.2) AND NOT %ML2500.1;

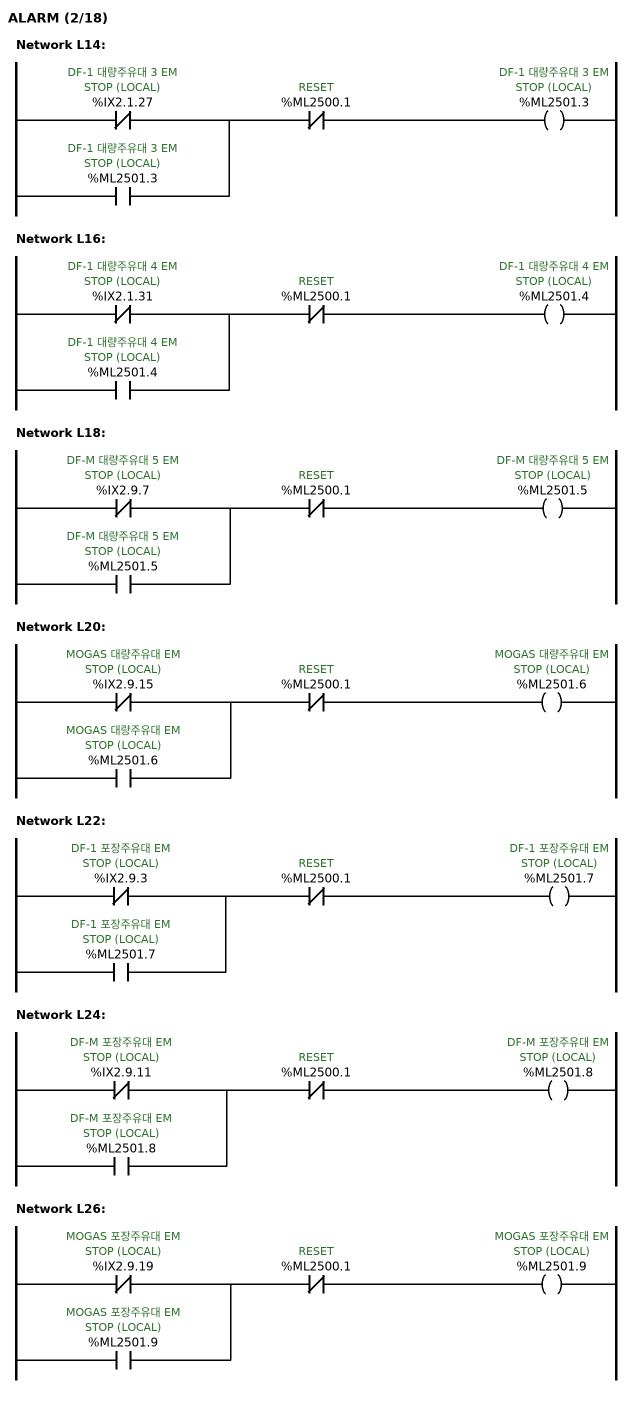
(* Rung L14 *)
%ML2501.3 := (NOT %IX2.1.27 OR %ML2501.3) AND NOT %ML2500.1;
(* Rung L16 *)
%ML2501.4 := (NOT %IX2.1.31 OR %ML2501.4) AND NOT %ML2500.1;
(* Rung L18 *)
%ML2501.5 := (NOT %IX2.9.7 OR %ML2501.5) AND NOT %ML2500.1;
(* Rung L20 *)
%ML2501.6 := (NOT %IX2.9.15 OR %ML2501.6) AND NOT %ML2500.1;
(* Rung L22 *)
%ML2501.7 := (NOT %IX2.9.3 OR %ML2501.7) AND NOT %ML2500.1;
(* Rung L24 *)
%ML2501.8 := (NOT %IX2.9.11 OR %ML2501.8) AND NOT %ML2500.1;
(* Rung L26 *)
%ML2501.9 := (NOT %IX2.9.19 OR %ML2501.9) AND NOT %ML2500.1;

